// TIA Portal V20 export
DATA_BLOCK "DB_AnalogInputDataPLC"   // DB1307
TITLE = TEMPERATURE SETTINGS
{ S7_Optimized_Access := 'FALSE'; DB_Accessible_From_OPC_UA := 'FALSE' }
AUTHOR : SAN
// stored: AutoNumber false, DBAccessibleFromOPCUA false, DBAccessibleFromWebserver false
   VAR RETAIN
      Laser_Power_Meter : "AnalogInDataPLC_DT";
      Axis_B_Clamping_Part : "AnalogInDataPLC_DT";
      Laser_Air_Pressure_Process : "AnalogInDataPLC_DT";
      Inlet_Air_Pressure : "AnalogInDataPLC_DT";
      Ambiant_Temperature : "AnalogInDataPLC_DT";
      Machine_Temperature : "AnalogInDataPLC_DT";
      Cold_Water_Temperature_Input : "AnalogInDataPLC_DT";
      Cold_Water_Temperature_Output : "AnalogInDataPLC_DT";
      X_Axis_Temperature_PT1000 : "AnalogInDataPLC_DT";
      Y_Axis_Temperature_PT1000 : "AnalogInDataPLC_DT";
      X_Axis_Temperature_PTC : "AnalogInDataPLC_DT";
      Y_Axis_Temperature_PTC : "AnalogInDataPLC_DT";
      Nozzle_Overpressure : "AnalogInDataPLC_DT";
      Optical_Path_Overpressure : "AnalogInDataPLC_DT";
      Laser_Head_Overpressure : "AnalogInDataPLC_DT";
      ZL_Axis_Overpressure : "AnalogInDataPLC_DT";
      XY_Axis_Overpressure : "AnalogInDataPLC_DT";
      Left_Aspiration : "AnalogInDataPLC_DT";
      Right_Aspiration : "AnalogInDataPLC_DT";
      Free_IW458 : "AnalogInDataPLC_DT";
      Clim_Temperature : "AnalogInDataPLC_DT";
      Free_IW482 : "AnalogInDataPLC_DT";
      Free_IW484 : "AnalogInDataPLC_DT";
      Free_IW486 : "AnalogInDataPLC_DT";
      Sensor_Controller_Station1 : "AnalogInDataPLC_DT";
      Cabinet_Temperature : "AnalogInDataPLC_DT";
      Free_IW464 : "AnalogInDataPLC_DT";
      Free_IW466 : "AnalogInDataPLC_DT";
   END_VAR
BEGIN
   Laser_Power_Meter.LimitUp := 10.0;
   Laser_Power_Meter.LimitDown := 0.0;
   Laser_Power_Meter.TypeProbe := 2;
   Axis_B_Clamping_Part.LimitUp := 27648.0;
   Axis_B_Clamping_Part.LimitDown := 0.0;
   Axis_B_Clamping_Part.TypeProbe := 2;
   Laser_Air_Pressure_Process.LimitUp := 10.0;
   Laser_Air_Pressure_Process.LimitDown := 0.0;
   Laser_Air_Pressure_Process.TypeProbe := 2;
   Laser_Air_Pressure_Process.EnableAlarmMin := True;
   Laser_Air_Pressure_Process.EnableWarningMin := True;
   Laser_Air_Pressure_Process.EnableWarningMax := True;
   Laser_Air_Pressure_Process.EnableAlarmMax := True;
   Inlet_Air_Pressure.LimitUp := 10.0;
   Inlet_Air_Pressure.LimitDown := 0.0;
   Inlet_Air_Pressure.TypeProbe := 2;
   Inlet_Air_Pressure.EnableAlarmMin := True;
   Inlet_Air_Pressure.EnableWarningMin := True;
   Inlet_Air_Pressure.EnableWarningMax := True;
   Inlet_Air_Pressure.EnableAlarmMax := True;
   Ambiant_Temperature.TypeProbe := 0;
   Ambiant_Temperature.EnableAlarmMin := True;
   Ambiant_Temperature.EnableWarningMin := True;
   Ambiant_Temperature.EnableWarningMax := True;
   Ambiant_Temperature.EnableAlarmMax := True;
   Machine_Temperature.TypeProbe := 0;
   Machine_Temperature.EnableAlarmMin := True;
   Machine_Temperature.EnableWarningMin := True;
   Machine_Temperature.EnableWarningMax := True;
   Machine_Temperature.EnableAlarmMax := True;
   Cold_Water_Temperature_Input.TypeProbe := 0;
   Cold_Water_Temperature_Input.EnableAlarmMin := True;
   Cold_Water_Temperature_Input.EnableWarningMin := True;
   Cold_Water_Temperature_Input.EnableWarningMax := True;
   Cold_Water_Temperature_Input.EnableAlarmMax := True;
   Cold_Water_Temperature_Output.TypeProbe := 0;
   Cold_Water_Temperature_Output.EnableAlarmMin := True;
   Cold_Water_Temperature_Output.EnableWarningMin := True;
   Cold_Water_Temperature_Output.EnableWarningMax := True;
   Cold_Water_Temperature_Output.EnableAlarmMax := True;
   X_Axis_Temperature_PT1000.TypeProbe := 1;
   X_Axis_Temperature_PT1000.EnableAlarmMin := True;
   X_Axis_Temperature_PT1000.EnableWarningMin := True;
   X_Axis_Temperature_PT1000.EnableWarningMax := True;
   X_Axis_Temperature_PT1000.EnableAlarmMax := True;
   Y_Axis_Temperature_PT1000.TypeProbe := 1;
   Y_Axis_Temperature_PT1000.EnableAlarmMin := True;
   Y_Axis_Temperature_PT1000.EnableWarningMin := True;
   Y_Axis_Temperature_PT1000.EnableWarningMax := True;
   Y_Axis_Temperature_PT1000.EnableAlarmMax := True;
   X_Axis_Temperature_PTC.TypeProbe := 6;
   Y_Axis_Temperature_PTC.TypeProbe := 6;
   Nozzle_Overpressure.LimitUp := 10.0;
   Nozzle_Overpressure.LimitDown := 0.0;
   Nozzle_Overpressure.TypeProbe := 2;
   Nozzle_Overpressure.EnableAlarmMin := True;
   Nozzle_Overpressure.EnableWarningMin := True;
   Nozzle_Overpressure.EnableWarningMax := True;
   Nozzle_Overpressure.EnableAlarmMax := True;
   Optical_Path_Overpressure.LimitUp := 10.0;
   Optical_Path_Overpressure.LimitDown := 0.0;
   Optical_Path_Overpressure.TypeProbe := 2;
   Optical_Path_Overpressure.EnableAlarmMin := True;
   Optical_Path_Overpressure.EnableWarningMin := True;
   Optical_Path_Overpressure.EnableWarningMax := True;
   Optical_Path_Overpressure.EnableAlarmMax := True;
   Laser_Head_Overpressure.LimitUp := 10.0;
   Laser_Head_Overpressure.LimitDown := 0.0;
   Laser_Head_Overpressure.TypeProbe := 2;
   Laser_Head_Overpressure.EnableAlarmMin := True;
   Laser_Head_Overpressure.EnableWarningMin := True;
   Laser_Head_Overpressure.EnableWarningMax := True;
   Laser_Head_Overpressure.EnableAlarmMax := True;
   ZL_Axis_Overpressure.LimitUp := 10.0;
   ZL_Axis_Overpressure.LimitDown := 0.0;
   ZL_Axis_Overpressure.TypeProbe := 2;
   ZL_Axis_Overpressure.EnableAlarmMin := True;
   ZL_Axis_Overpressure.EnableWarningMin := True;
   ZL_Axis_Overpressure.EnableWarningMax := True;
   ZL_Axis_Overpressure.EnableAlarmMax := True;
   XY_Axis_Overpressure.LimitUp := 10.0;
   XY_Axis_Overpressure.LimitDown := 0.0;
   XY_Axis_Overpressure.TypeProbe := 2;
   XY_Axis_Overpressure.EnableAlarmMin := True;
   XY_Axis_Overpressure.EnableWarningMin := True;
   XY_Axis_Overpressure.EnableWarningMax := True;
   XY_Axis_Overpressure.EnableAlarmMax := True;
   Left_Aspiration.LimitUp := 2000.0;
   Left_Aspiration.LimitDown := 0.0;
   Left_Aspiration.TypeProbe := 5;
   Left_Aspiration.EnableAlarmMin := True;
   Left_Aspiration.EnableWarningMin := True;
   Left_Aspiration.EnableWarningMax := True;
   Left_Aspiration.EnableAlarmMax := True;
   Right_Aspiration.LimitUp := 2000.0;
   Right_Aspiration.LimitDown := 0.0;
   Right_Aspiration.TypeProbe := 5;
   Right_Aspiration.EnableAlarmMin := True;
   Right_Aspiration.EnableWarningMin := True;
   Right_Aspiration.EnableWarningMax := True;
   Right_Aspiration.EnableAlarmMax := True;
   Clim_Temperature.TypeProbe := 0;
   Sensor_Controller_Station1.LimitUp := 10.0;
   Sensor_Controller_Station1.LimitDown := -10.0;
   Sensor_Controller_Station1.TypeProbe := 3;
   Cabinet_Temperature.LimitUp := 50.0;
   Cabinet_Temperature.LimitDown := 0.0;
   Cabinet_Temperature.TypeProbe := 2;
END_DATA_BLOCK
